// Mitsubishi GX Works2 project: 240528_링카운터조작패널2   PLC: Q03UDV

PROGRAM MAIN
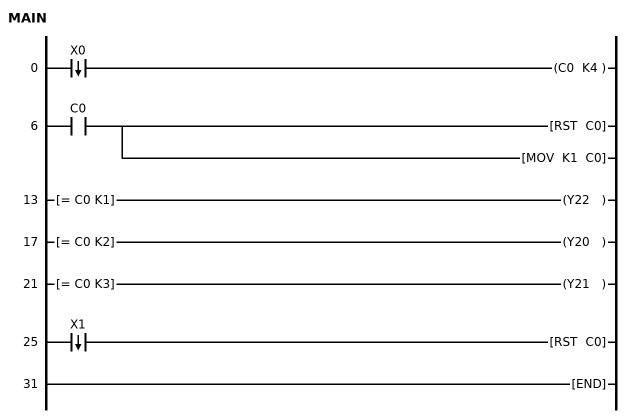
0     LDF     X0
      OUT     C0 K4
6     LD      C0
      RST     C0
      MOV     K1 C0
13    LD=     C0 K1
      OUT     Y22
17    LD=     C0 K2
      OUT     Y20
21    LD=     C0 K3
      OUT     Y21
25    LDF     X1
      RST     C0
31    END
END_PROGRAM
